(* Logix 5000 project; controller EsteiraSeletoraParte3 vendor 1 type 14 code 89 rev 20.11; software revision 20.05 *)

TASK MainTask (continuous, watchdog 500 ms) : MainProgram

MODULES
   Controller : vendor 1 type 14 code 89 (CompactLogixL23E_QBFC1_Controller 0, rev 20.11)
      LocalENB : vendor 1 type 12 code 191 (CompactLogixL23E_QBFC1_Ethernet 1, rev 20.11)
      Local : CompactBus (CompactVirtualAdapter 3, rev 20.11)
         Discrete_Inputs : vendor 1 type 7 code 320 (Compact 1, rev 3.1, Input RPI 20 ms)
         Discrete_Outputs : vendor 1 type 7 code 322 (Compact 2, rev 3.1, Output RPI 20 ms)
         Analog_IO : vendor 1 type 10 code 120 (Compact 3, rev 1.1, Output RPI 80 ms)
         Counters : vendor 1 type 109 code 70 (Compact 4, rev 1.1, Output RPI 20 ms)
END_MODULES

PROGRAM MainProgram   (* main routine MainRoutine *)

ROUTINE MainRoutine   (* ladder *)
END_ROUTINE
END_PROGRAM
